//{attribute 'qualified_only'}
VAR_GLOBAL
	Always_ON : BOOL := 1;
	Vacuum_Grants : ARRAY [0..31] OF BOOL;
	Vacuum_Requests : ARRAY [0..31] OF BOOL;
	Conv_Max_Times : ARRAY [0..31] OF DWORD := [32(30000)];
	Conv_Last_Times : ARRAY [0..31] OF DWORD;
END_VAR

(* stored: Version 1.1.0.1, ProductVersion 3.1.4024.13
   GVL GVL: Id {a9896aa3-c00d-4ec7-ba08-8202e16864e0} *)
